PROGRAM FlowUnits
VAR
END_VAR

PROPERTY Bar : string
GET
Bar := 'bar(g)';
END_GET
END_PROPERTY

PROPERTY PUBLIC LsMin : STRING
GET
LsMin := 'ls/min';
END_GET
END_PROPERTY

PROPERTY Sccm : STRING
GET
Sccm := 'sccm';
END_GET
END_PROPERTY

PROPERTY Slm : STRING
GET
Slm := 'slm';
END_GET
END_PROPERTY

END_PROGRAM

(* stored: Version 1.1.0.1, ProductVersion 3.1.4024.15
   POU FlowUnits: Id {e60bf494-1e97-08f8-3614-cad4ba620baa}, SpecialFunc None
   Property Bar: Id {055a85b4-d70f-09b0-028a-77151b32974b}
   Get Get: Id {4be92b17-c16c-061c-001e-2cf2baab53dd}
   Property LsMin: Id {950295d4-12c6-049e-3910-478a09487627}
   Get Get: Id {88032ad0-6141-0677-3988-0462e19c5af1}
   Property Sccm: Id {84400b5d-276f-0652-2fa2-da989247d2ba}
   Get Get: Id {7770c86f-d1e9-0036-3e37-ced778762d58}
   Property Slm: Id {af8ea509-426f-0f58-2412-d3b01988e582}
   Get Get: Id {a1cb2249-a064-066a-3e90-d8ec1e413158} *)
